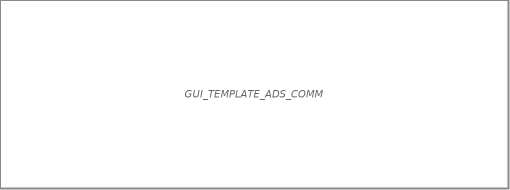
VISUALIZATION GUI_ADS_COMM_TEST  // 510x190
    Frame (0,0 508x188)
        shows GUI_TEMPLATE_ADS_COMM(m_Instance := MAIN.USB1)
END_VISUALIZATION

(* stored: Version 1.1.0.1, ProductVersion 3.1.4022.16
   Visu GUI_ADS_COMM_TEST: Id {5c721df8-2d32-43ea-8cce-8e48fd9bd61d} *)
